Fanuc KAREL source: ka00054.KL

PROGRAM KA00054
%NOLOCKGROUP
VAR
SRC : POSITION;DST : XYZWPR
BEGIN
--
DST=SRC
END KA00054
